(* CODESYS project TrafficControl.project
   Title: Traffic control simulator
   Version: 1.0
   Company: TK Automation
   Author: Toni Kucic

Project tree, tasks and I/O mapping:
  SoftPLC : CODESYS Control Win V3 x64, 3S - Smart Software Solutions GmbH, version 3.5.14.10
    application Application
      libraries: Standard, * (System); Util, * (System); Standard64, * (System); VisuDialogs, * (System)
      task VISU_TASK (cyclic, interval 50 ms, priority 31) calls VisuElems.Visu_Prg
      task xsim03 (cyclic, interval t#5ms, priority 1) calls xsim03
      task xc03_Task (cyclic, interval t#50ms, priority 1) calls xc03_TrafficControl
      image pool ImagePool
      IO/
        global variables xgv03
      Control/
        program xc03_TrafficControl [ST]
      Simulator/
        program xsim03 [ST]
      HMI/
        visualisation xv03_TrafficControl
  libraries: VisuSymbols, 3.5.10.0 (System)
  00000000-0000-0000-0000-000000000000|C:\Users\Toni\Google Drive\Projekti\PLC projekti\tkautomation school\Functional Descriptions\FD_TrafficControl.docx
  FD_TrafficControl
  5ce3da45-db07-42e7-a21c-a00fff4ed8f6|Car1.png
  text list GlobalTextList
  5ce3da45-db07-42e7-a21c-a00fff4ed8f6|trafficlightsystem.jpg
  5ce3da45-db07-42e7-a21c-a00fff4ed8f6|Car4.png
  5ce3da45-db07-42e7-a21c-a00fff4ed8f6|Car3.png
  5ce3da45-db07-42e7-a21c-a00fff4ed8f6|Car2.png
  5ce3da45-db07-42e7-a21c-a00fff4ed8f6|Car1.png
  5ce3da45-db07-42e7-a21c-a00fff4ed8f6|Projects\breaker1.jpg
  5ce3da45-db07-42e7-a21c-a00fff4ed8f6|Projects\breaker2.jpg
  5ce3da45-db07-42e7-a21c-a00fff4ed8f6|Projects\Ventilator1.jpg
  5ce3da45-db07-42e7-a21c-a00fff4ed8f6|Projects\Ventilator2.jpg
  5ce3da45-db07-42e7-a21c-a00fff4ed8f6|Projects\main-switchboard_1.jpg
  5ce3da45-db07-42e7-a21c-a00fff4ed8f6|Projects\breaker1.jpg
  5ce3da45-db07-42e7-a21c-a00fff4ed8f6|Projects\breaker2.jpg
  5ce3da45-db07-42e7-a21c-a00fff4ed8f6|Projects\cloud with rain.jpg
  5ce3da45-db07-42e7-a21c-a00fff4ed8f6|Car2.png
  function block CollisionDetection [ST]
  text list System
  5ce3da45-db07-42e7-a21c-a00fff4ed8f6|Car3.png
  5ce3da45-db07-42e7-a21c-a00fff4ed8f6|C:\Users\Toni\Google Drive\Projekti\PLC projekti\Materijali\traffic_light_05.jpgsmall.jpg
  5ce3da45-db07-42e7-a21c-a00fff4ed8f6|boom.png
  5ce3da45-db07-42e7-a21c-a00fff4ed8f6|Projects\Ventilator1small.jpg
  5ce3da45-db07-42e7-a21c-a00fff4ed8f6|Projects\Ventilator2small.jpg
  5ce3da45-db07-42e7-a21c-a00fff4ed8f6|Projects\igrasatasterima.JPG
  5ce3da45-db07-42e7-a21c-a00fff4ed8f6|Projects\empty-road-intersection-icon-cartoon-style-H67GFG.jpg
  5ce3da45-db07-42e7-a21c-a00fff4ed8f6|Projects\traffic_light_05.jpgsmall.jpg
  5ce3da45-db07-42e7-a21c-a00fff4ed8f6|Projects\breaker1.jpg
  5ce3da45-db07-42e7-a21c-a00fff4ed8f6|Projects\breaker2.jpg
  5ce3da45-db07-42e7-a21c-a00fff4ed8f6|C:\Users\Toni\Google Drive\Projekti\PLC projekti\Materijali\traffic_light_05.jpgsmall.jpg
  function block MoveSprite [ST]
  5ce3da45-db07-42e7-a21c-a00fff4ed8f6|boom.png
  5ce3da45-db07-42e7-a21c-a00fff4ed8f6|bottle_empty.png
  5ce3da45-db07-42e7-a21c-a00fff4ed8f6|bottle_broken.png
  5ce3da45-db07-42e7-a21c-a00fff4ed8f6|bottle_halffull.png
  5ce3da45-db07-42e7-a21c-a00fff4ed8f6|bottle_full.png
  5ce3da45-db07-42e7-a21c-a00fff4ed8f6|roller1.png
  5ce3da45-db07-42e7-a21c-a00fff4ed8f6|roller2.png
  5ce3da45-db07-42e7-a21c-a00fff4ed8f6|cranebackground.png
  5ce3da45-db07-42e7-a21c-a00fff4ed8f6|cranemover.png
  5ce3da45-db07-42e7-a21c-a00fff4ed8f6|hook.png
  5ce3da45-db07-42e7-a21c-a00fff4ed8f6|trafficlightsystem.jpg
  5ce3da45-db07-42e7-a21c-a00fff4ed8f6|Car4.png
*)

// SoftPLC/Application/IO/xgv03
{attribute 'qualified_only'}
VAR_GLOBAL
	
	//Configuration
	cfgPeriodTime: TIME := T#84S;
	cfgStartDirection: DINT := 0;
 
	//Inputs
	(* No inputs *)
	
	//Outputs
	TLight1Red : BOOL;	(* DIGITAL OUTPUT	Activate red light traffic light 1 *)
	TLight1Yellow : BOOL;	(* DIGITAL OUTPUT	Activate yellow light traffic light 1 *)
	TLight1Green : BOOL;	(* DIGITAL OUTPUT	Activate green light traffic light 1 *)
	TLight2Red : BOOL;	(* DIGITAL OUTPUT	Activate red light traffic light 2 *)
	TLight2Yellow : BOOL;	(* DIGITAL OUTPUT	Activate yellow light traffic light 2 *)
	TLight2Green : BOOL;	(* DIGITAL OUTPUT	Activate green light traffic light 2 *)
	TLight3Red : BOOL;	(* DIGITAL OUTPUT	Activate red light traffic light 3 *)
	TLight3Yellow : BOOL;	(* DIGITAL OUTPUT	Activate yellow light traffic light 3 *)
	TLight3Green : BOOL;	(* DIGITAL OUTPUT	Activate green light traffic light 3 *)
	TLight4Red : BOOL;	(* DIGITAL OUTPUT	Activate red light traffic light 4 *)
	TLight4Yellow : BOOL;	(* DIGITAL OUTPUT	Activate yellow light traffic light 4 *)
	TLight4Green : BOOL;	(* DIGITAL OUTPUT	Activate green light traffic light 4 *)

END_VAR

// SoftPLC/Application/Simulator/xsim03
PROGRAM xsim03
VAR
	Car1X: INT := 925; (* Red car *)
	Car1Y: INT := 740;
	Car1Width: INT := 100;
	Car1Height: INT := 230;
	Car2X: INT := 420; (* Blue car *)
	Car2Y: INT := 511;
	Car2Width: INT := 230;
	Car2Height: INT := 100;
	Car3X : INT := 1160; (* Green car *)
	Car3Y: INT := 366;
	Car3Width: INT := 230;
	Car3Height: INT := 100;
	Car4X: INT := 775; (* Yellow car *)
	Car4Y: INT := 0;
	Car4Width: INT := 100;
	Car4Height: INT := 230;
	Speed : INT := 1;
	vCarCrash: BOOL;
	vReset: BOOL;
	xExplosion: INT;
	yExplosion: INT;
	
	Car3Car4Coll: CollisionDetection;
	Car3Car1Coll: CollisionDetection;
	Car2Car1Coll: CollisionDetection;
	Car2Car4Coll: CollisionDetection;

	MoveCar1: MoveSprite;
	MoveCar2: MoveSprite;
	MoveCar3: MoveSprite;
	MoveCar4: MoveSprite;
END_VAR

(* Collision detection *)
(* Car3 and Car 4 *)
Car3Car4Coll(
	xcor1:= Car3X, 
	ycor1:= Car3Y, 
	height1:= Car3Height, 
	width1:= Car3Width, 
	xcor2:= Car4X, 
	ycor2:= Car4Y, 
	height2:= Car4Height, 
	width2:= Car4Width);
(* Car3 and Car 1 *)
Car3Car1Coll(
	xcor1:= Car3X, 
	ycor1:= Car3Y, 
	height1:= Car3Height, 
	width1:= Car3Width, 
	xcor2:= Car1X, 
	ycor2:= Car1Y, 
	height2:= Car1Height, 
	width2:= Car1Width);
(* Car2 and Car 4 *)
Car2Car4Coll(
	xcor1:= Car2X, 
	ycor1:= Car2Y, 
	height1:= Car2Height, 
	width1:= Car2Width, 
	xcor2:= Car4X, 
	ycor2:= Car4Y, 
	height2:= Car4Height, 
	width2:= Car4Width);
(* Car2 and Car 1 *)
Car2Car1Coll(
	xcor1:= Car2X, 
	ycor1:= Car2Y, 
	height1:= Car2Height, 
	width1:= Car2Width, 
	xcor2:= Car1X, 
	ycor2:= Car1Y, 
	height2:= Car1Height, 
	width2:= Car1Width);

IF Car3Car4Coll.isCollision OR Car3Car1Coll.isCollision OR Car2Car4Coll.isCollision OR Car2Car1Coll.isCollision THEN
	vCarCrash := TRUE;
ELSE
	vCarCrash := FALSE;	
END_IF

(* Explosion graphic *)
IF Car3Car4Coll.isCollision THEN
	xExplosion := Car3X;
	yExplosion := Car3Y;
ELSIF Car3Car1Coll.isCollision THEN
	xExplosion := Car3X;
	yExplosion := Car3Y;
ELSIF Car2Car4Coll.isCollision THEN
	xExplosion := Car2X + Car2Width;
	yExplosion := Car2Y;
ELSIF Car2Car1Coll.isCollision THEN
	xExplosion := Car2X + Car2Width;
	yExplosion := Car2Y;
ELSE
	xExplosion := 2000;
	yExplosion := 2000;
END_IF

(* Car movements *)
IF  vCarCrash THEN
	//wait
	IF vReset THEN
		(* Reset to start position *)
		Car1X:= 925;
		Car1Y:= 740;
		Car2X:= 420;
		Car2Y:= 511;
		Car3X:= 1160;
		Car3Y:= 366;
		Car4X:= 775;
		Car4Y:= 0;
	END_IF
ELSE
	(* Define what cars do depending on lights *)
	(* car moves if its green for him or he is past the traffic ligght but stops at the traffic light if its red, or yellow.*)
	IF xgv03.TLight4Green OR Car1Y - 740 < 0 OR Car1Y - 740 > Speed THEN
		MoveCar1(
		xCor:= Car1X, 
		yCor:= Car1Y, 
		xScreen:= 1830, 
		yScreen:= 930,
		SpriteWidth:= Car1Width, 
		SpriteHeight:= Car1Height, 
		ySpeed:= -Speed, 
		xSpeed:= 0 );
	END_IF;
	IF xgv03.TLight2Green OR Car2X - 420 < 0 OR Car2X - 420 > Speed THEN
		MoveCar2(
		xCor:= Car2X, 
		yCor:= Car2Y, 
		xScreen:= 1830, 
		yScreen:= 930,
		SpriteWidth:= Car2Width, 
		SpriteHeight:= Car2Height,  
		ySpeed:= 0, 
		xSpeed:= Speed );
	END_IF;
	IF xgv03.TLight1Green OR Car3X - 1160 < 0 OR Car3X - 1160 > Speed THEN
		MoveCar3(
		xCor:= Car3X, 
		yCor:= Car3Y, 
		xScreen:= 1830, 
		yScreen:= 930,
		SpriteWidth:= Car3Width, 
		SpriteHeight:= Car3Height,  
		ySpeed:= 0, 
		xSpeed:= -Speed );
	END_IF;
	IF xgv03.TLight3Green OR Car4Y - 0 < 0 OR Car4Y - 0 > Speed THEN
		MoveCar4(
		xCor:= Car4X, 
		yCor:= Car4Y, 
		xScreen:= 1830, 
		yScreen:= 930,
		SpriteWidth:= Car4Width, 
		SpriteHeight:= Car4Height,  
		ySpeed:= Speed, 
		xSpeed:= 0 );
	END_IF;
END_IF

END_PROGRAM

// CollisionDetection
FUNCTION_BLOCK CollisionDetection
VAR_INPUT
	xcor1: REAL := 0; (* X Coordinate of object 1 *)
	ycor1: REAL := 0; (* Y Coordinate of object 1 *)
	height1: REAL := 0; (* Height of object 1 *)
	width1: REAL := 0;	(* Width of object 1 *)
	xcor2: REAL := 0; (* X Coordinate of object 2 *)
	ycor2: REAL := 0; (* Y Coordinate of object 2 *)
	height2: REAL := 0; (* Height of object 1 *)
	width2: REAL := 0;	(* Width of object 1 *)	
END_VAR
VAR_OUTPUT
	isCollision: BOOL := FALSE;
END_VAR
VAR
END_VAR

IF xcor1 < (xcor2 + width2) AND
   (xcor1 + width1) > xcor2 AND
   ycor1 < (ycor2 + height2) AND
  ( height1 + ycor1) > ycor2 THEN
   isCollision := TRUE;
ELSE
	isCollision := FALSE;
END_IF

END_FUNCTION_BLOCK

// MoveSprite
FUNCTION_BLOCK MoveSprite
VAR_IN_OUT
	xCor : INT := 0;
	yCor : INT := 0;
END_VAR
VAR_INPUT
	xScreen: INT := 0; (* Width of the screen *)
	yScreen: INT := 0; (* Height of the screen *)
	SpriteWidth: INT := 0; (* Width of the sprite *)
	SpriteHeight: INT := 0; (* Height of the sprite *)	
	ySpeed: INT :=0; (* Control up or down movement with +- *)
	xSpeed: INT :=0; (* Control left or right movement with +- *)
END_VAR
VAR
END_VAR

(* Reseting the position if sprite goes off screen *)
(* If moving left to right *)
IF xCor >= xScreen  AND xSpeed > 0 THEN
	xCor := -SpriteWidth;
(* If moving right to left *)
ELSIF xCor <= -SpriteWidth AND xSpeed < 0 THEN
	xCor := xScreen;	
END_IF
(* If moving from up, down *)
IF yCor >= yScreen AND ySpeed > 0 THEN
	yCor := -SpriteHeight;
(* If moving from down, up *)
ELSIF yCor < -SpriteHeight AND ySpeed < 0 THEN
	yCor := yScreen;	
END_IF

(* Actual moving of the coordinates *)
xCor := xCor + xSpeed;
yCor := yCor + ySpeed;

END_FUNCTION_BLOCK

// SoftPLC/Application/Control/xc03_TrafficControl
PROGRAM xc03_TrafficControl
VAR
	vSequenceA: DINT:=1;
	TimerA:TOF;
	vSequenceB: DINT:=0;
	TimerB:TOF;
	Start: BOOL;
	StartOld: BOOL;
	vSequence: DINT := 0;
	TactTimer : TON;
	vPeriodTime: TIME := T#85S;
	vElapsedTime: TIME;
END_VAR


TactTimer(IN:=TRUE, PT:=vPeriodTime, ET => vElapsedTime);
IF TactTimer.Q THEN
	TactTimer(IN:=FALSE);
END_IF
(* Direction Up, Down traffic light *)
xgv03.TLight3Red := vElapsedTime <= T#5S OR vElapsedTime >= T#37S AND vElapsedTime <= T#85S;
xgv03.TLight3Yellow := vElapsedTime > T#3S AND vElapsedTime <= T#5S OR vElapsedTime >= T#35S AND vElapsedTime <= T#37S;
xgv03.TLight3Green := vElapsedTime >= T#5S AND vElapsedTime <= T#35S;

(* Mirror the other side of the Up, Down direction *)
xgv03.TLight4Red := xgv03.TLight3Red;
xgv03.TLight4Yellow := xgv03.TLight3Yellow;
xgv03.TLight4Green := xgv03.TLight3Green;

(* Direction Left, Right traffic light *)
xgv03.TLight2Red := vElapsedTime >= T#0S AND vElapsedTime <= T#39S OR vElapsedTime >= T#71S AND vElapsedTime <= T#85S;
xgv03.TLight2Yellow := vElapsedTime > T#37S AND vElapsedTime <= T#39S OR vElapsedTime >= T#69S AND vElapsedTime <= T#71S;
xgv03.TLight2Green := vElapsedTime >= T#39S AND vElapsedTime <= T#69S;

(* Mirror the other side of the Left, Right direction *)
xgv03.TLight1Red := xgv03.TLight2Red;
xgv03.TLight1Yellow := xgv03.TLight2Yellow;
xgv03.TLight1Green := xgv03.TLight2Green;
(*CASE vSequence OF
	0:
	(* Starting sequence, direction Up, Down *)
	TimerA
	Task03GVL.TLight1Red := TRUE;
	
END_CASE
CASE vSequenceA OF
	0: TimerA(IN:=FALSE,PT:=T#20S);
	Task03GVL.TLight1Yellow:= FALSE;
	Task03GVL.TLight1Red:= FALSE;
	Task03GVL.TLight1Green:= TimerA.Q;
	Task03GVL.TLight2Green := Task03GVL.TLight1Green;
	IF NOT TimerA.Q THEN
		TimerA(IN:=TRUE);
		vSequenceA:=1;
	END_IF
	1: TimerA(IN:=FALSE,PT:=T#4S);
	Task03GVL.TLight1Red:= FALSE;
	Task03GVL.TLight1Green:= FALSE;
	Task03GVL.TLight1Yellow:= TimerA.Q;
	Task03GVL.TLight2Yellow := Task03GVL.TLight1Yellow;
	IF NOT TimerA.Q THEN
		TimerA(IN:=TRUE);
		vSequenceA:=2;
	END_IF
		2: TimerA(IN:=FALSE,PT:=T#30S);
	Task03GVL.TLight1Green:= FALSE;
	Task03GVL.TLight1Yellow:= FALSE;
	Task03GVL.TLight1Red:= TimerA.Q;
	Task03GVL.TLight2Red := Task03GVL.TLight1Red;
	IF NOT TimerA.Q THEN
		TimerA(IN:=TRUE);
		vSequenceA:=3;
	END_IF
		3: TimerA(IN:=FALSE,PT:=T#4S);
	Task03GVL.TLight1Green:= FALSE;
	Task03GVL.TLight1Red:= TimerA.Q;
	Task03GVL.TLight1Yellow:= TimerA.Q;
	Task03GVL.TLight2Red := Task03GVL.TLight1Red;
	Task03GVL.TLight2Yellow := Task03GVL.TLight1Yellow;
	IF NOT TimerA.Q THEN
		TimerA(IN:=TRUE);
		vSequenceA:=0;
		IF vSequenceB=6 THEN
		vSequenceB:=3;	
		END_IF
		
	END_IF
END_CASE

CASE vSequenceB OF
	0: TimerB(IN:=FALSE,PT:=T#4S);
	Task03GVL.TLight3Green:= FALSE;
	Task03GVL.TLight3Red:= TimerB.Q;
	Task03GVL.TLight3Yellow:= TimerB.Q;
	Task03GVL.TLight4Red := Task03GVL.TLight3Red;
	Task03GVL.TLight4Yellow := Task03GVL.TLight3Yellow;
	IF NOT TimerB.Q THEN
		TimerB(IN:=TRUE);
		vSequenceB:=1;
	END_IF
	
	1: TimerB(IN:=FALSE,PT:=T#20S);
	Task03GVL.TLight3Yellow:= FALSE;
	Task03GVL.TLight3Red:= FALSE;
	Task03GVL.TLight3Green:= TimerB.Q;
	Task03GVL.TLight4Green := Task03GVL.TLight3Green;
	IF NOT TimerB.Q THEN
		TimerB(IN:=TRUE);
		vSequenceB:=2;
	END_IF
	
	2: TimerB(IN:=FALSE,PT:=T#4S);
	Task03GVL.TLight3Red:= FALSE;
	Task03GVL.TLight3Green:= FALSE;
	Task03GVL.TLight3Yellow:= TimerB.Q;
	Task03GVL.TLight4Yellow := Task03GVL.TLight3Yellow;
	IF NOT TimerB.Q THEN
		TimerB(IN:=TRUE);
		vSequenceB:=3;
	END_IF
	
		3: TimerB(IN:=FALSE,PT:=T#30S);
	Task03GVL.TLight3Green:= FALSE;
	Task03GVL.TLight3Yellow:= FALSE;
	Task03GVL.TLight3Red:= TimerB.Q;
	Task03GVL.TLight4Red := Task03GVL.TLight3Red;
	IF NOT TimerB.Q THEN
		TimerB(IN:=TRUE);
		vSequenceB:=0;
	END_IF
		
END_CASE
END_IF;*)

END_PROGRAM

// SoftPLC/Application/HMI/xv03_TrafficControl
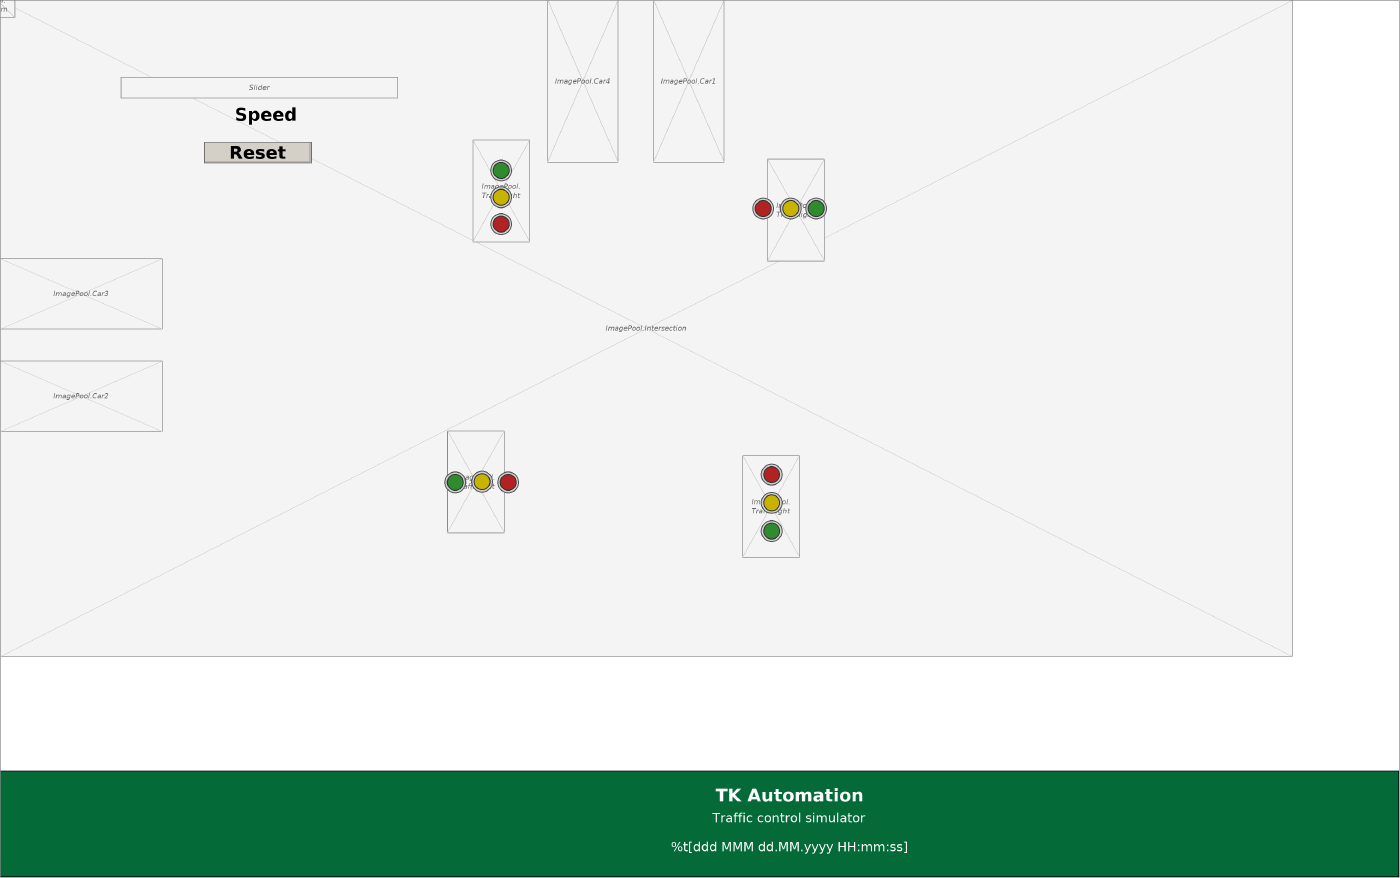
VISUALIZATION xv03_TrafficControl  // 1982x1244
    Image (0,0 1830x930), image: ImagePool.Intersection
    Image (1051,645 81x145), image: ImagePool.Trafficlight
    Image (1086,225 81x145), angle 270, image: ImagePool.Trafficlight
    Image (633,610 81x145), angle 90, image: ImagePool.Trafficlight
    Image (669,198 81x145), angle 179, image: ImagePool.Trafficlight
    Lamp1 (1075,655 35x35), variable: xgv03.TLight4Red, style: Lamp-Lamp1-Red
    Lamp1 (1075,735 35x35), variable: xgv03.TLight4Green, style: Lamp-Lamp1-Green
    Lamp1 (1075,695 35x35), variable: xgv03.TLight4Yellow, style: Lamp-Lamp1-Yellow
    Lamp1 (702,666 35x35), variable: xgv03.TLight2Red, style: Lamp-Lamp1-Red
    Lamp1 (627,666 35x35), variable: xgv03.TLight2Green, style: Lamp-Lamp1-Green
    Lamp1 (665,665 35x35), variable: xgv03.TLight2Yellow, style: Lamp-Lamp1-Yellow
    Lamp1 (1063,278 35x35), variable: xgv03.TLight1Red, style: Lamp-Lamp1-Red
    Lamp1 (1102,278 35x35), variable: xgv03.TLight1Yellow, style: Lamp-Lamp1-Yellow
    Lamp1 (1138,278 35x35), variable: xgv03.TLight1Green, style: Lamp-Lamp1-Green
    Lamp1 (692,224 35x35), variable: xgv03.TLight3Green, style: Lamp-Lamp1-Green
    Lamp1 (692,300 35x35), variable: xgv03.TLight3Red, style: Lamp-Lamp1-Red
    Lamp1 (692,262 35x35), variable: xgv03.TLight3Yellow, style: Lamp-Lamp1-Yellow
    Image (925,0 100x230), image: ImagePool.Car1
        p2738717112: xsim03.Car1Y
    Image (775,0 100x230), image: ImagePool.Car4
        p2738717112: xsim03.Car4Y
    Image (0,366 230x100), image: ImagePool.Car3
        p3560616238: xsim03.Car3X
    Image (0,511 230x100), image: ImagePool.Car2
        p3560616238: xsim03.Car2X
    Slider (171,109 392x30), variable: xsim03.Speed, scale 1..5
    Label (210,147 333x30), "Speed"
    Image (-29,-25 50x50), image: ImagePool.Boom
        p3560616238: xsim03.xExplosion
        p2738717112: xsim03.yExplosion
    Button (289,201 152x30), "Reset", invisible if: NOT xsim03.vCarCrash
        tap xsim03.vReset
    Rectangle (16,1209 1830x30)
    Rectangle (0,1092 1980x150)
    Label (962,1110 312x33), "TK Automation"
    Label (367,1144 1500x30), "Traffic control simulator"
    Rectangle (826,1185 584x30), "%t[ddd MMM dd.MM.yyyy HH:mm:ss]"
END_VISUALIZATION

(* text list System (id | default)
  Apr | Apr
  April | April
  Aug | Aug
  August | August
  Dec | Dec
  December | December
  Feb | Feb
  February | February
  Fri | Fri
  Friday | Friday
  Jan | Jan
  January | January
  Jul | Jul
  July | July
  Jun | Jun
  June | June
  Mar | Mar
  March | March
  May | May
  May_3Letter | May
  Mon | Mon
  Monday | Monday
  Nov | Nov
  November | November
  Oct | Oct
  October | October
  Sat | Sat
  Saturday | Saturday
  Sep | Sep
  September | September
  Sun | Sun
  Sunday | Sunday
  Thu | Thu
  Thursday | Thursday
  Tue | Tue
  Tuesday | Tuesday
  Wed | Wed
  Wednesday | Wednesday
   |  *)
